FUNCTION_BLOCK "Cinta de Volcado (Máquina)"   // FB8, LAD
TITLE = Bloque Máquina para las cintas de volcado
{ S7_Optimized_Access := 'TRUE' }
VERSION : 0.1
// Incluye estados de defecto por tiempo límite, mal arranque y  emergencia. Se ha considerado una señal de rearme que devuelve a la máquina al reposo desde la emergencia. Para volver desde el defecto se ha configurado un aviso que puede ser desactivado por el usuario (una vez se ha solucionado el problema).
// Esta máquina se encarga de volcar  las piezas que expulsa cada CNC (una vez terminado el tratamiento), evitando colisiones en la cinta de evacuación (que es común a las tres CNCs).
// Se hará uso del bloque "Cinta de Volcado (Aviso de Disponibilidad)", que mediante una señal de aviso indicará cuándo es seguro incoporar una pieza a la cinta.
// NOTA: es importante diferenciar la cinta de evacuación (común a las tres CNCs) y la cinta de volcado que conecta cada máquina con la anterior.
// (EMPLEA EL BLOQUE AUXILIAR FB7 "Aviso de Disponibilidad")
   VAR_INPUT
      Start : Bool;   // Señal de arranque de la máquina
      EMER : Bool;   // Señal de emergencia
      S2 : Bool;   // Sensor de presencia al final de la cinta de volcado.
      S3_izquierdo : Bool;   // Sensor de la cinta de evacuación, a la izquierda de la intersección con la cinta de volcado.
      S3_derecho : Bool;   // Sensor de la cinta de evacuación, a la derecha de la intersección con la cinta de volcado.
      señal_fin_tratamiento : Bool;   // Aviso de que la operación de corte/serigrafía ha concluido exitosamente
      Rearme : Bool;   // Señal de rearme de la máquina
      tiempo_seguridad : Time;   // Tiempo de seguridad para considerar intersección libre
      tiempo_límite_volcado : Time;   // Tiempo límite para transportar la pieza hasta el límite de la cinta de volcado
      flag_sentido_cinta_inferior : Bool;   // Vale 1 cuando la cinta de evacuación se mueve de izquierda a derecha
   END_VAR
   VAR_OUTPUT
      MOTOR_V : Bool;   // Actuador que controla la cinta de volcado
      aviso_standby : Bool;   // Aviso de que la máquina está en standby
   END_VAR
   VAR_IN_OUT
      aviso_defecto : Bool;
   END_VAR
   VAR
      bit_de_trabajo : Bool;   // bit de trabajo para el arranque
      X_Standby : Bool;   // Estado de Standby
      X_Defecto_Tiempo : Bool;   // Estado de defecto de tiempo
      X_Defecto_Emergencia : Bool;   // Estado de defecto por emergencia
      X_Defecto_Posición : Bool;   // Estado de defecto por mal posicionamiento inicial
      X1 : Bool;   // Estado de trabajo. Se lleva la pieza hasta el borde de la cinta de volcado.
      X2 : Bool;   // Estado de comprobación. Cuando la cinta de evacuación esté libre, se incorpora la pieza.
      M_flanco_rearme : Bool;   // Marca de flanco de la señal rearme
      M_flanco_defecto : Bool;   // Marca de flanco para el aviso de defecto
      temporizador : TON_TIME;
      Aviso_de_Disponibilidad : "Cinta de Volcado (Aviso de Disponibilidad)";
      M_flanco_señal_fin_de_tratamiento : Bool;   // Marca de flanco para la señal de fin de tratamiento
   END_VAR
   VAR_TEMP
      aviso_interno_intersección_libre : Bool;   // Aviso interno que indica que es seguro incorporar una pieza.
   END_VAR
   VAR_TEMP   // added for the SCL form of the ladder/FBD networks
      _w1 : Bool;
   END_VAR
BEGIN

REGION Network 1 (STL): DESCONEXIÓN (Start:=False)
   // Aagado de la máquina, máxima prioridad. Se llama a las maniobras con RESET:=TRUE (en caso de haberlas).
   // Tan solo se ponen a cero las salidas, los estados internos se inicializarán en el arranque.
   // En este caso, "Aviso_de_Disponibilidad" no maneja actuadores y no acaba de cumplir el prototipo "maniobra".
         AN    #Start;
         JCN   _DESCONEXION;
         CALL  #Aviso_de_Disponibilidad
         ( S_izquierda                 := ,
           S_derecha                   := ,
           tiempo_limite               := ,
           RESET                       := TRUE,
           flag_sentido_cinta_inferior := ,
           aviso_intersección_libre    := #aviso_interno_intersección_libre
         );
         AN    #Start;
         R     #bit_de_trabajo;
         R     #aviso_standby;
         R     #MOTOR_V;
         R     #aviso_defecto;
         BEC;
   _DESCONEXION:NOP   0;
END_REGION

REGION Network 2 (STL): Llamada al bloque auxiliar FB7 "Aviso de Disponibilidad"
         A     #Start;
         JCN   _CALL_AVISO_DISPONIBILIDAD;
         CALL  #Aviso_de_Disponibilidad
         ( S_izquierda                 := #S3_izquierdo,
           S_derecha                   := #S3_derecho,
           tiempo_limite               := #tiempo_seguridad,
           RESET                       := FALSE,
           flag_sentido_cinta_inferior := #flag_sentido_cinta_inferior,
           aviso_intersección_libre    := #aviso_interno_intersección_libre
         );
   _CALL_AVISO_DISPONIBILIDAD:NOP   0;
END_REGION

REGION Network 3 (STL): DEFECTO (emergencia)
   // Defecto prioritario. LLamamos a las maniobras con RESET:=TRUE (en caso de haberlas)
         A     #EMER;
         JCN   _EMER;
         CALL  #Aviso_de_Disponibilidad
         ( S_izquierda                 := ,
           S_derecha                   := ,
           tiempo_limite               := ,
           RESET                       := TRUE,
           flag_sentido_cinta_inferior := ,
           aviso_intersección_libre    := #aviso_interno_intersección_libre
         );
         A     #EMER;
         S     #X_Defecto_Emergencia;
         R     #X_Standby;
         R     #X_Defecto_Tiempo;
         R     #X_Defecto_Posición;
         R     #X1;
         R     #X2;
   _EMER:NOP   0;
END_REGION

REGION Network 4 (STL): DEFECTO (tiempo excedido durante la expansión)
   // Ante el aviso de defecto por tiempo (lo proporciona el bloque maniobra) se accede al estado de defecto.
         A     #X1;
         A     #temporizador.Q;
         S     #X_Defecto_Tiempo;
         R     #X1;
END_REGION

REGION Network 5 (STL): DEFECTO (mal posicionamiento en el arranque)
   // Si al arrancar, la máquina no está posicionada correctamente, se accede al correspondiente estado de defecto. 
   // Se ha considerado que un mal posicionamiento en el arranque sería S2==TRUE. Esto podría suceder si una pieza ha permanecido en la cinta de volcado frente al sensor.
         A     #X_Standby;
         A     #S2;
         S     #X_Defecto_Posición;
         R     #X_Standby;
END_REGION

REGION Network 6 (STL): Aviso de defecto (para el rearme)
   // Se avisará al usuario cuando la máquina haya entrado en defecto
         A     #X_Defecto_Posición;
         O     #X_Defecto_Tiempo;
         FP    #M_flanco_defecto;
         S     #aviso_defecto;
END_REGION

REGION Network 7 (STL): REARME (emergencia)
   // Una vez se ha solucionado el problema  se vuelve al reposo con el flanco positivo de la señal rearme.
         A     #Rearme;
         FP    #M_flanco_rearme;
         A     #X_Defecto_Emergencia;
         AN    #EMER;
         S     #X_Standby;
         R     #X_Defecto_Emergencia;
END_REGION

REGION Network 8: REARME (Defecto de tiempo o posición)
   // Una vez se ha solucionado el problema, se vuelve al reposo al desactivarse el aviso de error (por el usuario)
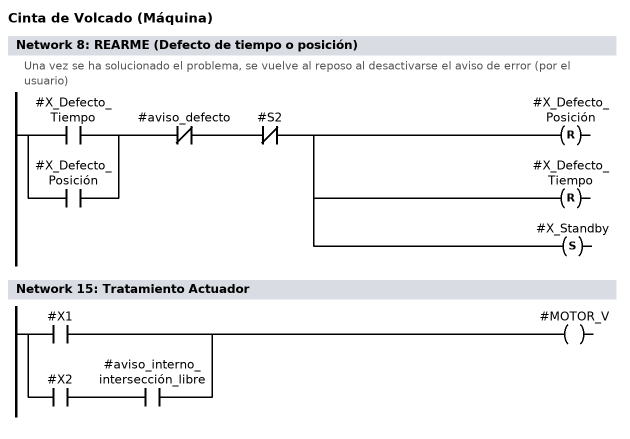
   RUNG wire#powerrail
      Contact( #X_Defecto_Tiempo )
      wire#w1
      I_Contact( #aviso_defecto )
      I_Contact( #S2 )
      wire#w2
      R_Coil( #X_Defecto_Posición )
   END_RUNG
   RUNG wire#powerrail
      Contact( #X_Defecto_Posición )
   END_RUNG wire#w1
   RUNG wire#w2
      R_Coil( #X_Defecto_Tiempo )
   END_RUNG
   RUNG wire#w2
      S_Coil( #X_Standby )
   END_RUNG
   // the same network as SCL:
   #_w1 := (#X_Defecto_Tiempo OR #X_Defecto_Posición) AND NOT #aviso_defecto AND NOT #S2;
   IF #_w1 THEN
       #X_Defecto_Posición := FALSE;
       #X_Defecto_Tiempo := FALSE;
       #X_Standby := TRUE;
   END_IF;
END_REGION

REGION Network 9 (STL): ARRANQUE
   // Arrancamos la máquina, inicializando el estado de standby (X0)
         A     #Start;
         FP    #bit_de_trabajo;
         S     #X_Standby;
         R     #X_Defecto_Tiempo;
         R     #X_Defecto_Emergencia;
         R     #X_Defecto_Posición;
         R     #M_flanco_defecto;
         R     #M_flanco_rearme;
         R     #X1;
         R     #X2;
         R     #aviso_interno_intersección_libre;
END_REGION

REGION Network 10 (STL): Configuración Temporizador
   // Se empleará un TON (sin memoria) para el defecto de tiempo. Saltará si la pieza no llega al final de la cinta de volcado en el tiempo especificado.
         CALL  #temporizador
         ( IN := #X1,
           PT := #tiempo_límite_volcado,
           Q  := ,
           ET :=
         );
END_REGION

REGION Network 11 (STL): X_Standby ->X1
   // Cuando se recibe el aviso de que la CNC ha concluido el tratamiento, se pone en acción la cinta de volcado.
         A     #señal_fin_tratamiento;
         FP    #M_flanco_señal_fin_de_tratamiento;
         A     #X_Standby;
         R     #X_Standby;
         S     #X1;
END_REGION

REGION Network 12 (STL): X1->X2
   // Al alcanzar la pieza el final de la cinta (S2==TRUE), se accede al estado de comprobación.
         A     #X1;
         A     #S2;
         R     #X1;
         S     #X2;
END_REGION

REGION Network 13 (STL): X2->X_Standby
   // Al abandonar la pieza la cinta de volcado (S2==FALSE), se vuelve al estado de espera.
         A     #X2;
         AN    #S2;
         R     #X2;
         S     #X_Standby;
END_REGION

REGION Network 14 (STL): Aviso de Standby (para el usuario)
   // Avisa de que la máquina está en standby y funcionando correctamente
         A     #X_Standby;
         =     #aviso_standby;
END_REGION

REGION Network 15: Tratamiento Actuador
   RUNG wire#powerrail
      Contact( #X1 )
      wire#w1
      Coil( #MOTOR_V )
   END_RUNG
   RUNG wire#powerrail
      Contact( #X2 )
      Contact( #aviso_interno_intersección_libre )
   END_RUNG wire#w1
   // the same network as SCL:
   #MOTOR_V := #X1 OR (#X2 AND #aviso_interno_intersección_libre);
END_REGION
END_FUNCTION_BLOCK

// folder: Máquinas/Sistemas

FUNCTION_BLOCK "Sistema de Alimentación"   // FB1, LAD
TITLE = Sistema de Alimentación
{ S7_Optimized_Access := 'TRUE' }
VERSION : 0.1
// Incluye los tres pistones de alimentación de piezas.  Su finalidad es englobar los tres pistones de alimentación en un solo bloque haciendo uso de multi-instancia.
// (BLOQUE NO AUTOCONTENIDO)
   VAR
      Pistón_Corte : "Pistón (Máquina)";
      Pistón_Laminado : "Pistón (Máquina)";
      Pistón_Serigrafiado : "Pistón (Máquina)";
   END_VAR
BEGIN

REGION Network 1 (STL): Llamada Incondicional
         CALL  #Pistón_Corte
         ( Start                := "X_MA1",
           EMER                 := "X21",
           SC                   := "FC1_C",
           SE                   := "FC1_E",
           Rearme               := "X20",
           pieza_detectada      := "SC0",
           pieza_válida         := "pieza_válida_corte",
           tiempo_expansión     := "DATOS_PRODUCCION".tiempo_exp,
           tiempo_compresión    := "DATOS_PRODUCCION".tiempo_comp,
           aviso_CNC_disponible := "aviso_Standby_máquina_corte",
           EXP                  := "EXP1",
           COMP                 := "COMP1",
           aviso_standby        := "aviso_Standby_pistón1",
           aviso_defecto        := "aviso_Defecto_pistón1"
         );
         CALL  #Pistón_Laminado
         ( Start                := "X_MA2",
           EMER                 := "X21",
           SC                   := "FC2_C",
           SE                   := "FC2_E",
           Rearme               := "X20",
           pieza_detectada      := "SL0",
           pieza_válida         := "pieza_válida_laminado",
           tiempo_expansión     := "DATOS_PRODUCCION".tiempo_exp,
           tiempo_compresión    := "DATOS_PRODUCCION".tiempo_comp,
           aviso_CNC_disponible := "aviso_Standby_máquina_laminado",
           EXP                  := "EXP2",
           COMP                 := "COMP2",
           aviso_standby        := "aviso_Standby_pistón2",
           aviso_defecto        := "aviso_Defecto_pistón2"
         );
         CALL  #Pistón_Serigrafiado
         ( Start                := "X_MA3",
           EMER                 := "X21",
           SC                   := "FC3_C",
           SE                   := "FC3_E",
           Rearme               := "X20",
           pieza_detectada      := "SS0",
           pieza_válida         := "pieza_válida_serigrafía",
           tiempo_expansión     := "DATOS_PRODUCCION".tiempo_exp,
           tiempo_compresión    := "DATOS_PRODUCCION".tiempo_comp,
           aviso_CNC_disponible := "aviso_Standby_máquina_serigrafiado",
           EXP                  := "EXP3",
           COMP                 := "COMP3",
           aviso_standby        := "aviso_Standby_pistón3",
           aviso_defecto        := "aviso_Defecto_pistón3"
         );
END_REGION
END_FUNCTION_BLOCK

FUNCTION_BLOCK "Sistema de Volcado"   // FB9, LAD
TITLE = Sistema de Volcado
{ S7_Optimized_Access := 'TRUE' }
VERSION : 0.1
// Incluye las tres cintas de volcado de piezas. Su finalidad es englobar las tres cintas de volcado en un solo bloque haciendo uso de multi-instancia.
// (BLOQUE NO AUTOCONTENIDO)
   VAR
      Cinta_Volcado_Corte : "Cinta de Volcado (Máquina)";
      Cinta_Volcado_Laminado : "Cinta de Volcado (Máquina)";
      Cinta_Volcado_Serigrafiado : "Cinta de Volcado (Máquina)";
   END_VAR
BEGIN

REGION Network 1 (STL): Llamada Incondicional
         CALL  #Cinta_Volcado_Corte
         ( Start                       := "X_ME1",
           EMER                        := "X21",
           S2                          := "SC2",
           S3_izquierdo                := "SC3_Izquierda",
           S3_derecho                  := "SC3_Derecha",
           señal_fin_tratamiento       := "aviso_fin_tratamiento_corte",
           Rearme                      := "X20",
           tiempo_seguridad            := "DATOS_PRODUCCION".tiempo_evacuación,
           tiempo_límite_volcado       := "DATOS_PRODUCCION".tiempo_volcado,
           flag_sentido_cinta_inferior := "DATOS_PRODUCCION".flag_sentido_cinta_inferior,
           MOTOR_V                     := "CINTA_VOLCADO_Corte",
           aviso_standby               := "aviso_Standby_cinta1",
           aviso_defecto               := "aviso_Defecto_cinta1"
         );
         CALL  #Cinta_Volcado_Laminado
         ( Start                       := "X_ME2",
           EMER                        := "X21",
           S2                          := "SL2",
           S3_izquierdo                := "SL3_Izquierda",
           S3_derecho                  := "SL3_Derecha",
           señal_fin_tratamiento       := "aviso_fin_tratamiento_laminado",
           Rearme                      := "X20",
           tiempo_seguridad            := "DATOS_PRODUCCION".tiempo_evacuación,
           tiempo_límite_volcado       := "DATOS_PRODUCCION".tiempo_volcado,
           flag_sentido_cinta_inferior := "DATOS_PRODUCCION".flag_sentido_cinta_inferior,
           MOTOR_V                     := "CINTA_VOLCADO_Laminado",
           aviso_standby               := "aviso_Standby_cinta2",
           aviso_defecto               := "aviso_Defecto_cinta2"
         );
         CALL  #Cinta_Volcado_Serigrafiado
         ( Start                       := "X_ME3",
           EMER                        := "X21",
           S2                          := "SS2",
           S3_izquierdo                := "SS3_Izquierda",
           S3_derecho                  := "SS3_Derecha",
           señal_fin_tratamiento       := "aviso_fin_tratamiento_serigrafiado",
           Rearme                      := "X20",
           tiempo_seguridad            := "DATOS_PRODUCCION".tiempo_evacuación,
           tiempo_límite_volcado       := "DATOS_PRODUCCION".tiempo_volcado,
           flag_sentido_cinta_inferior := "DATOS_PRODUCCION".flag_sentido_cinta_inferior,
           MOTOR_V                     := "CINTA_VOLCADO_Serigrafiado",
           aviso_standby               := "aviso_Standby_cinta3",
           aviso_defecto               := "aviso_Defecto_cinta3"
         );
END_REGION
END_FUNCTION_BLOCK

// folder: Tests

FUNCTION "test_unitario_maniobra_pistón" : Void   // FC1, LAD
TITLE = TEST UNITARIO maniobra simple con error por sobrepasamiento de tiempo límite y RESET
{ S7_Optimized_Access := 'TRUE' }
VERSION : 0.1
// test passed (Si)
BEGIN

REGION Network 1 (STL): Llamada a la maniobra
   // Ejecuta la maniobra una vez y desenclava la señal de disparo. Mediante observación se 
   // puede ver qué aviso ha quedado activo.
         A     "Tag_1";
         JCN   _TEST_MAN1;
         CALL  "Pistón (Maniobra Simple)", "Pistón (Maniobra Simple)_test_DB"
         ( SFIN                      := "Tag_2",
           tiempo_limite             := "DATOS_PRODUCCION".tiempo_exp,
           RESET                     := "Tag_3",
           ACT                       := "Tag_4",
           aviso_error_tiempo_limite := "Tag_5",
           aviso_fin_maniobra        := "Tag_6"
         );
         A     "Tag_5";
         O     "Tag_6";
         R     "Tag_1";
   _TEST_MAN1:NOP   0;
END_REGION
END_FUNCTION

FUNCTION "test_unitario_maquina_pistón" : Void   // FC2, LAD
TITLE = TEST UNITARIO de una máquina del control
{ S7_Optimized_Access := 'TRUE' }
VERSION : 0.1
// TEST UNITARIO de una máquina del control
BEGIN

REGION Network 1: Llamada inconcicional al bloque
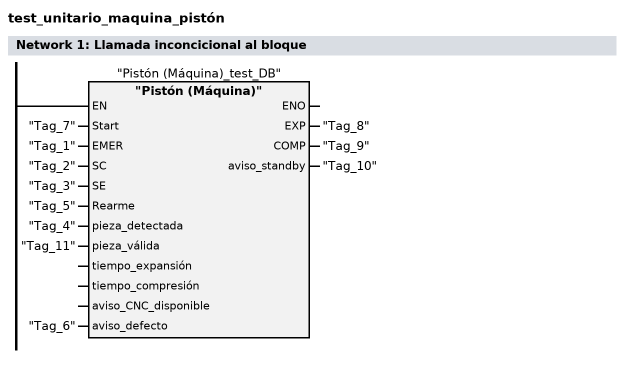
   RUNG wire#powerrail
      "Pistón (Máquina)_test_DB"(Start := "Tag_7", EMER := "Tag_1", SC := "Tag_2", SE := "Tag_3", Rearme := "Tag_5", pieza_detectada := "Tag_4", pieza_válida := "Tag_11", aviso_defecto := "Tag_6", EXP => "Tag_8", COMP => "Tag_9", aviso_standby => "Tag_10", tiempo_expansión :=, tiempo_compresión :=, aviso_CNC_disponible :=)
   END_RUNG
   // the same network as SCL:
   "Pistón (Máquina)_test_DB"(Start := "Tag_7",   // "Pistón (Máquina)"
                           EMER := "Tag_1",
                           SC := "Tag_2",
                           SE := "Tag_3",
                           Rearme := "Tag_5",
                           pieza_detectada := "Tag_4",
                           pieza_válida := "Tag_11",
                           aviso_defecto := "Tag_6",
                           EXP => "Tag_8",
                           COMP => "Tag_9",
                           aviso_standby => "Tag_10");
END_REGION
END_FUNCTION

FUNCTION "test_unitario_máquina_laminado" : Void   // FC6, LAD
TITLE = TEST UNITARIO de una máquina del control
{ S7_Optimized_Access := 'TRUE' }
VERSION : 0.1
// test_passed (SI)
BEGIN

REGION Network 1: Llamada inconcicional al bloque
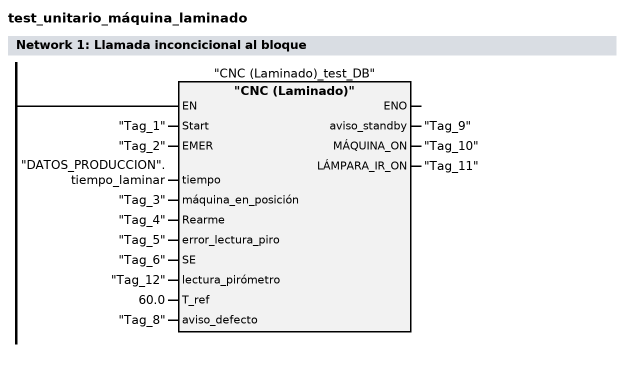
   RUNG wire#powerrail
      "CNC (Laminado)_test_DB"(Start := "Tag_1", EMER := "Tag_2", tiempo := "DATOS_PRODUCCION".tiempo_laminar, máquina_en_posición := "Tag_3", Rearme := "Tag_4", error_lectura_piro := "Tag_5", SE := "Tag_6", lectura_pirómetro := "Tag_12", T_ref := 60.0, aviso_defecto := "Tag_8", aviso_standby => "Tag_9", MÁQUINA_ON => "Tag_10", LÁMPARA_IR_ON => "Tag_11")
   END_RUNG
   // the same network as SCL:
   "CNC (Laminado)_test_DB"(Start := "Tag_1",   // "CNC (Laminado)"
                           EMER := "Tag_2",
                           tiempo := "DATOS_PRODUCCION".tiempo_laminar,
                           máquina_en_posición := "Tag_3",
                           Rearme := "Tag_4",
                           error_lectura_piro := "Tag_5",
                           SE := "Tag_6",
                           lectura_pirómetro := "Tag_12",
                           T_ref := 60.0,
                           aviso_defecto := "Tag_8",
                           aviso_standby => "Tag_9",
                           MÁQUINA_ON => "Tag_10",
                           LÁMPARA_IR_ON => "Tag_11");
END_REGION
END_FUNCTION

FUNCTION "test_unitario_máquina_corte" : Void   // FC7, LAD
TITLE = TEST UNITARIO de una máquina del control
{ S7_Optimized_Access := 'TRUE' }
VERSION : 0.1
// test_passed (SI)
BEGIN

REGION Network 1: Llamada incondicional
   // IMPORTANTE: Antes de cualquier rearme, la máquina tiene que estar en su posición inicial (máquina_en_posición:=TRUE)
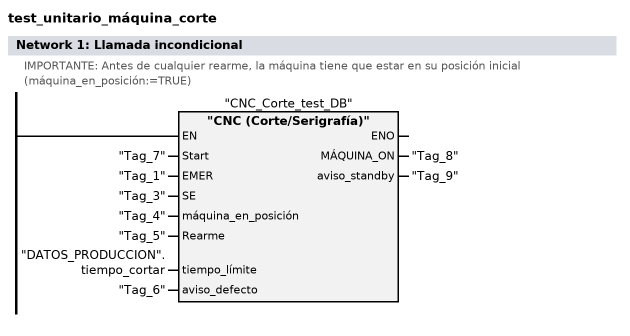
   RUNG wire#powerrail
      "CNC_Corte_test_DB"(Start := "Tag_7", EMER := "Tag_1", SE := "Tag_3", máquina_en_posición := "Tag_4", Rearme := "Tag_5", tiempo_límite := "DATOS_PRODUCCION".tiempo_cortar, aviso_defecto := "Tag_6", MÁQUINA_ON => "Tag_8", aviso_standby => "Tag_9")
   END_RUNG
   // the same network as SCL:
   "CNC_Corte_test_DB"(Start := "Tag_7",   // "CNC (Corte/Serigrafía)"
                       EMER := "Tag_1",
                       SE := "Tag_3",
                       máquina_en_posición := "Tag_4",
                       Rearme := "Tag_5",
                       tiempo_límite := "DATOS_PRODUCCION".tiempo_cortar,
                       aviso_defecto := "Tag_6",
                       MÁQUINA_ON => "Tag_8",
                       aviso_standby => "Tag_9");
END_REGION
END_FUNCTION

FUNCTION "test_unitario_máquina_brazo" : Void   // FC9, LAD
TITLE = TEST UNITARIO de una máquina del control
{ S7_Optimized_Access := 'TRUE' }
VERSION : 0.1
// test_passed (SI)
BEGIN

REGION Network 1: Llamada inconcicional al bloque
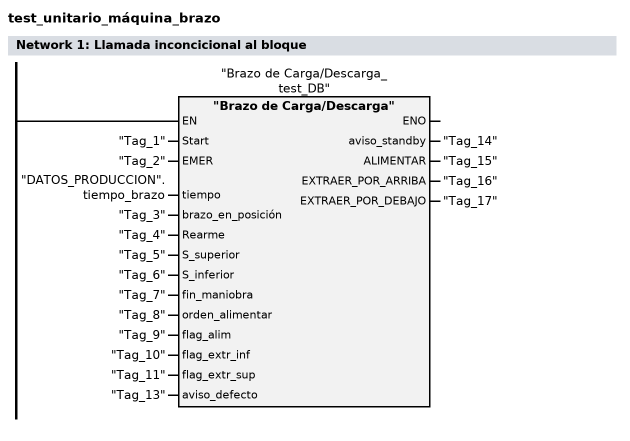
   RUNG wire#powerrail
      "Brazo de Carga/Descarga_test_DB"(Start := "Tag_1", EMER := "Tag_2", tiempo := "DATOS_PRODUCCION".tiempo_brazo, brazo_en_posición := "Tag_3", Rearme := "Tag_4", S_superior := "Tag_5", S_inferior := "Tag_6", fin_maniobra := "Tag_7", orden_alimentar := "Tag_8", flag_alim := "Tag_9", flag_extr_inf := "Tag_10", flag_extr_sup := "Tag_11", aviso_defecto := "Tag_13", aviso_standby => "Tag_14", ALIMENTAR => "Tag_15", EXTRAER_POR_ARRIBA => "Tag_16", EXTRAER_POR_DEBAJO => "Tag_17")
   END_RUNG
   // the same network as SCL:
   "Brazo de Carga/Descarga_test_DB"(Start := "Tag_1",   // "Brazo de Carga/Descarga"
                           EMER := "Tag_2",
                           tiempo := "DATOS_PRODUCCION".tiempo_brazo,
                           brazo_en_posición := "Tag_3",
                           Rearme := "Tag_4",
                           S_superior := "Tag_5",
                           S_inferior := "Tag_6",
                           fin_maniobra := "Tag_7",
                           orden_alimentar := "Tag_8",
                           flag_alim := "Tag_9",
                           flag_extr_inf := "Tag_10",
                           flag_extr_sup := "Tag_11",
                           aviso_defecto := "Tag_13",
                           aviso_standby => "Tag_14",
                           ALIMENTAR => "Tag_15",
                           EXTRAER_POR_ARRIBA => "Tag_16",
                           EXTRAER_POR_DEBAJO => "Tag_17");
END_REGION
END_FUNCTION

FUNCTION "test_unitario_disponibilidad_cinta_de_evacuación" : Void   // FC10, LAD
TITLE = TEST UNITARIO sub-proceso de monitorización de la cinta de evacuación
{ S7_Optimized_Access := 'TRUE' }
VERSION : 0.1
// test passed (Si)
BEGIN

REGION Network 1: Llamada a la maniobra
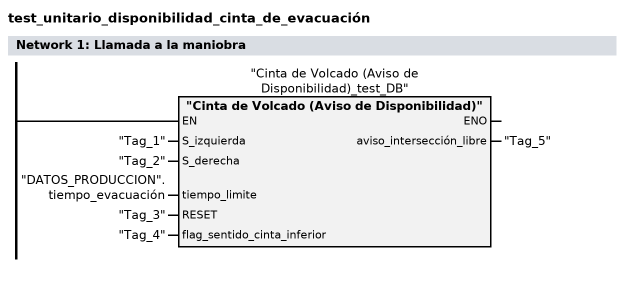
   RUNG wire#powerrail
      "Cinta de Volcado (Aviso de Disponibilidad)_test_DB"(S_izquierda := "Tag_1", S_derecha := "Tag_2", tiempo_limite := "DATOS_PRODUCCION".tiempo_evacuación, RESET := "Tag_3", flag_sentido_cinta_inferior := "Tag_4", aviso_intersección_libre => "Tag_5")
   END_RUNG
   // the same network as SCL:
   "Cinta de Volcado (Aviso de Disponibilidad)_test_DB"(S_izquierda := "Tag_1",   // "Cinta de Volcado (Aviso de Disponibilidad)"
                           S_derecha := "Tag_2",
                           tiempo_limite := "DATOS_PRODUCCION".tiempo_evacuación,
                           RESET := "Tag_3",
                           flag_sentido_cinta_inferior := "Tag_4",
                           aviso_intersección_libre => "Tag_5");
END_REGION
END_FUNCTION

FUNCTION "test_unitario_máquina_cinta_de_volcado" : Void   // FC11, LAD
{ S7_Optimized_Access := 'TRUE' }
VERSION : 0.1
BEGIN

REGION Network 1
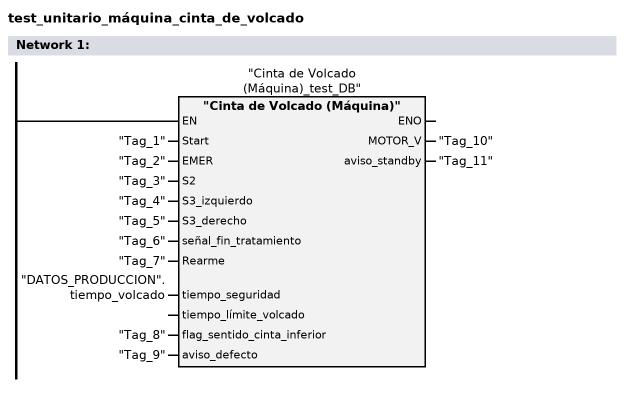
   RUNG wire#powerrail
      "Cinta de Volcado (Máquina)_test_DB"(Start := "Tag_1", EMER := "Tag_2", S2 := "Tag_3", S3_izquierdo := "Tag_4", S3_derecho := "Tag_5", señal_fin_tratamiento := "Tag_6", Rearme := "Tag_7", tiempo_seguridad := "DATOS_PRODUCCION".tiempo_volcado, flag_sentido_cinta_inferior := "Tag_8", aviso_defecto := "Tag_9", MOTOR_V => "Tag_10", aviso_standby => "Tag_11", tiempo_límite_volcado :=)
   END_RUNG
   // the same network as SCL:
   "Cinta de Volcado (Máquina)_test_DB"(Start := "Tag_1",   // "Cinta de Volcado (Máquina)"
                           EMER := "Tag_2",
                           S2 := "Tag_3",
                           S3_izquierdo := "Tag_4",
                           S3_derecho := "Tag_5",
                           señal_fin_tratamiento := "Tag_6",
                           Rearme := "Tag_7",
                           tiempo_seguridad := "DATOS_PRODUCCION".tiempo_volcado,
                           flag_sentido_cinta_inferior := "Tag_8",
                           aviso_defecto := "Tag_9",
                           MOTOR_V => "Tag_10",
                           aviso_standby => "Tag_11");
END_REGION
END_FUNCTION